FUNCTION_BLOCK ABSTRACT PolarisationFilterBase EXTENDS TExecution IMPLEMENTS IDevice
VAR_INPUT
END_VAR
VAR_OUTPUT
END_VAR
VAR
	{attribute 'OPC.UA.DA' := '0'}
	_name : STRING;
	{attribute 'OPC.UA.DA' := '0'}
	_deviceID : STRING;					
	{attribute 'OPC.UA.DA' := '0'}
	_family : DeviceFamily;			
	{attribute 'OPC.UA.DA' := '0'}
	_logger : Logger;
	{attribute 'OPC.UA.DA' := '0'}
	_message : StringBuilder;
	{attribute 'OPC.UA.DA' := '0'}
	_polarisationFilterConfig : DeviceConfiguration;
END_VAR

PROPERTY DeviceID : STRING
GET
DeviceID := _deviceID;
END_GET
SET
_deviceID := DeviceID;
END_SET
END_PROPERTY

PROPERTY Family : DeviceFamily
GET
Family := _family;
END_GET
SET
_family := Family;
END_SET
END_PROPERTY

METHOD PROTECTED ABSTRACT GetPosition 
VAR_INPUT
END_VAR
END_METHOD

METHOD PROTECTED ABSTRACT JogBackwardPosition
VAR_INPUT
	Execute : BOOL;
END_VAR
END_METHOD

METHOD PROTECTED ABSTRACT JogForwardPosition
VAR_INPUT
	Execute : BOOL;
END_VAR
END_METHOD

METHOD PROTECTED ABSTRACT MoveAbsPosition
VAR_INPUT
	Execute : BOOL;
	Position : LREAL;
END_VAR
END_METHOD

PROPERTY Name : STRING
GET
Name := _name;
END_GET
SET
_name := Name;
END_SET
END_PROPERTY

END_FUNCTION_BLOCK

(* stored: Version 1.1.0.1, ProductVersion 3.1.4024.3
   POU PolarisationFilterBase: Id {068f2ca3-fcd9-4644-b52e-278c2c90b1af}, SpecialFunc None
   Property DeviceID: Id {af91a433-4663-45bc-8e3a-c7138b85094d}
   Get Get: Id {58de6ac1-b8cb-426d-9277-42ce2005d2fc}
   Set Set: Id {b35b31cc-e767-407d-86f0-5140dca65838}
   Property Family: Id {8987b731-bee2-4c15-96ce-36df74ea4fe3}
   Get Get: Id {4425f55c-ecf4-4cac-9721-7eb5ac08ce15}
   Set Set: Id {7cb07c35-b3f0-4d7c-b738-9ae9eb22bdcf}
   Method GetPosition: Id {79894dfb-bac7-4fbf-ba7c-d93121d51e98}
   Method JogBackwardPosition: Id {43a934b4-4492-4cdc-b2e9-46b7080013bc}
   Method JogForwardPosition: Id {815c4111-de0d-464e-912a-13649f254091}
   Method MoveAbsPosition: Id {39178ee9-b62c-45f8-86ff-0ed6f705d3d5}
   Property Name: Id {c1040452-b13a-463e-afb1-31374684dd5a}
   Get Get: Id {abe9bbbb-0b29-454d-afd0-fbec79026c8d}
   Set Set: Id {13b23b6d-9ea2-4ad0-8c0a-e4622287719f} *)
